(* PLC project  *)

PROGRAM P
  VAR  (* added by the conversion: wires and edge detectors of the diagram *)
    _ADD2_ENO : BOOL;
    _ADD2_OUT : ANY;
  END_VAR

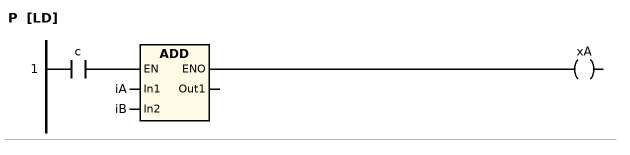
(* LD diagram, written out as Structured Text *)
_ADD2_OUT := ADD(EN := c, IN1 := iA, IN2 := iB, ENO => _ADD2_ENO);
xA := _ADD2_ENO;
END_PROGRAM
